FUNCTION Convert_ULINT_TO_DWORD : BOOL
VAR_INPUT
	in : ULINT;
	out : REFERENCE TO DWORD;
END_VAR
VAR
	converted : DWORD;
END_VAR

converted := ULINT_TO_DWORD(in);

IF (DWORD_TO_ULINT(converted) <> in) THEN
	RETURN;
END_IF

out := converted;
Convert_ULINT_TO_DWORD := TRUE;

END_FUNCTION

(* stored: Version 1.1.0.1, ProductVersion 3.1.4024.12
   POU Convert_ULINT_TO_DWORD: Id {055db101-08c5-497d-b00f-092bbc39da48}, SpecialFunc None *)
